Yaskawa INFORM job: blower_cylinder_program.JBI

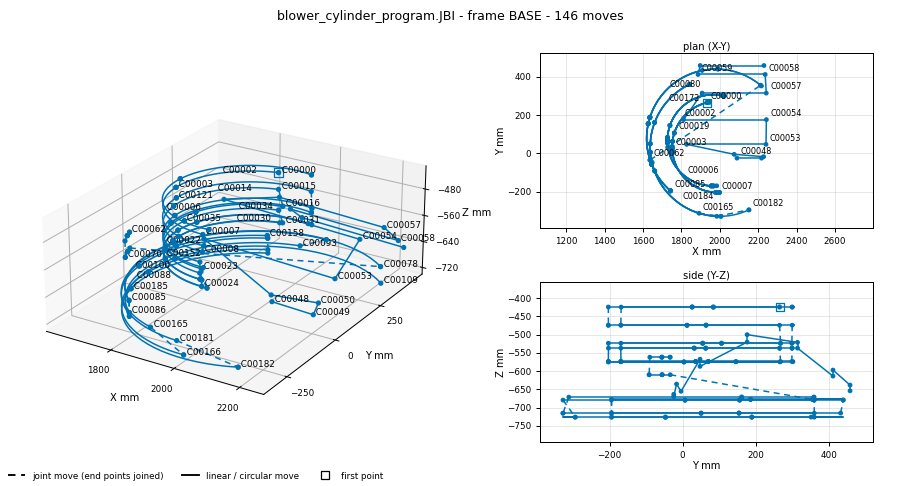
[picture p0: tool path of blower_cylinder_program.JBI in frame BASE, 146 of 201 moves have a stored position in this frame; points joined in program order, loops and branches not executed]
/JOB
//NAME blower_cylinder_program
//POS
///NPOS 190,0,190,0,0,0
///TOOL 0
///POSTYPE BASE
///RECTAN
///RCONF 0,0,0,0,0,0,0,0,0,0,0,0,0,0,0,0,0,0,0,0,0,0,0,0
C00000=1933.494064,265.432065,-424.583000,103.550681,-90.000000,5.000000
C00001=1933.494064,265.432065,-424.583000,103.550681,-90.000000,5.000000
C00002=1798.542139,176.350935,-424.583000,143.306547,-89.999999,5.000000
C00003=1751.564327,26.089320,-424.583000,-175.000000,-90.000000,5.000000
C00004=1751.564327,26.089320,-424.583000,-175.000000,-90.000000,5.000000
C00005=1751.564327,26.089320,-424.583000,-175.000000,-90.000000,5.000000
C00006=1811.478144,-123.700155,-424.583000,-138.369256,-90.000000,5.000000
C00007=1986.712740,-203.504840,-424.583000,-90.601327,-89.999999,5.000000
C00008=1985.205000,-203.484234,-474.602000,-90.964662,-90.000000,5.000000
C00009=1985.205000,-203.484234,-474.602000,-90.964662,-90.000000,5.000000
C00010=1831.755761,-143.919254,-474.602000,-131.465158,-89.999999,5.000000
C00011=1752.467395,12.011979,-474.602000,-174.629726,-90.000000,5.000000
C00012=1752.467395,12.011979,-474.602000,-174.629726,-90.000000,5.000000
C00013=1752.467395,12.011979,-474.602000,-174.629726,-90.000000,5.000000
C00014=1789.907703,163.961680,-474.602000,146.945900,-90.000000,5.000000
C00015=1933.747591,265.493022,-474.602000,103.487851,-90.000000,5.000000
C00016=1946.318295,268.151177,-523.863500,100.391501,-90.000000,5.000000
C00017=1946.318295,268.151177,-523.863500,100.391501,-90.000000,5.000000
C00018=1857.013607,231.918088,-523.863500,123.775687,-90.000000,5.000000
C00019=1762.672230,106.536544,-523.863500,162.306197,-90.000000,5.000000
C00020=1762.672230,106.536544,-523.863500,162.306197,-90.000000,5.000000
C00021=1762.672230,106.536544,-523.863500,162.306197,-90.000000,5.000000
C00022=1803.833605,-114.655285,-523.863500,-141.223119,-90.000000,5.000000
C00023=1981.181892,-203.382432,-523.863500,-91.934378,-90.000000,5.000000
C00024=1982.070197,-203.410772,-573.993000,-91.720226,-89.999999,5.000000
C00025=1982.070197,-203.410772,-573.993000,-91.720226,-89.999999,5.000000
C00026=1827.997866,-140.526698,-573.993000,-132.685079,-90.000000,5.000000
C00027=1751.426860,35.497028,-573.993000,175.000000,-90.000000,5.000000
C00028=1751.426860,35.497028,-573.993000,175.000000,-90.000000,5.000000
C00029=1751.426860,35.497028,-573.993000,175.000000,-90.000000,5.000000
C00030=1823.986848,205.273668,-573.993000,134.014193,-90.000000,5.000000
C00031=1946.357863,268.158430,-573.993000,100.381809,-89.999999,5.000000
C00032=1934.436096,265.657079,-537.267460,175.000000,-60.000000,-76.682693
C00033=1934.436096,265.657079,-537.267460,175.000000,-60.000000,-76.682693
C00034=1828.865200,209.855997,-537.267460,-175.000000,-60.000000,-47.598579
C00035=1753.185183,63.156372,-537.267460,175.000000,-60.000000,-6.978408
C00036=1753.185183,63.156372,-537.267460,175.000000,-60.000000,-6.978408
C00037=1753.185183,63.156372,-537.267460,175.000000,-60.000000,-6.978408
C00038=1809.805430,-121.797856,-537.267460,-175.000000,-60.000000,41.020368
C00039=1976.108054,-203.156798,-537.267460,-175.000000,-60.000000,86.841815
C00040=1998.571162,-203.333530,-575.058960,175.000000,-60.000000,92.256633
C00041=1998.571162,-203.333530,-575.058960,175.000000,-60.000000,92.256633
C00042=1843.618470,-153.736326,-575.058960,175.000000,-60.000000,52.245744
C00043=1753.406955,3.619432,-575.058960,175.000000,-60.000000,7.405254
C00044=1753.406955,3.619432,-575.058960,175.000000,-60.000000,7.405254
C00045=1753.406955,3.619432,-575.058960,175.000000,-60.000000,7.405254
C00046=1795.171150,171.711596,-575.058960,175.000000,-60.000000,-35.311600
C00047=1937.779187,266.423001,-575.058960,-175.000000,-60.000000,-77.509111
C00048=2089.306045,-24.353058,-663.745553,175.000000,-60.000000,90.065286
C00049=2217.470262,-24.353051,-669.800856,175.000000,-60.000000,90.065286
C00050=2228.297277,-16.748565,-635.673601,-175.000000,-60.000000,91.170202
C00051=2074.711330,-4.438705,-655.515790,175.000000,-66.623448,91.170202
C00052=1827.048359,47.582539,-567.652515,175.000000,-44.740427,92.732701
C00053=2240.740165,47.582562,-587.197981,175.000000,-44.740427,92.732701
C00054=2242.656280,176.551574,-520.760389,-170.133186,5.000000,5.000000
C00055=1810.757184,176.551550,-500.354693,-170.133186,5.000000,5.000000
C00056=1907.631611,314.643219,-521.482904,156.457092,5.000000,-5.000000
C00057=2242.006831,314.643237,-537.280944,156.457092,5.000000,-5.000000
C00058=2236.445037,411.851577,-613.890742,175.000000,-53.159924,-92.028486
C00059=1886.225138,411.851557,-597.344097,175.000000,-53.159924,-92.028486
C00060=1897.676258,458.517871,-638.458617,175.000000,-60.000000,-90.549119
C00061=2229.933616,458.517890,-654.156596,175.000000,-60.000000,-90.549119
C00062=1636.254154,-34.391820,-562.117000,-161.880193,-90.000000,5.000000
C00063=1636.254154,-34.391820,-562.117000,-161.880193,-90.000000,5.000000
C00064=1640.360805,-46.242627,-562.117000,-159.894424,-89.999999,5.000000
C00065=1644.466194,-56.930864,-562.117000,-158.081660,-90.000000,5.000000
C00066=1644.466194,-56.930864,-562.117000,-158.081660,-90.000000,5.000000
C00067=1644.466194,-56.930864,-562.117000,-158.081660,-90.000000,5.000000
C00068=1652.539385,-75.480262,-562.117000,-154.878428,-90.000000,5.000000
C00069=1659.732185,-89.968706,-562.117000,-152.317297,-89.999999,5.000000
C00070=1660.669780,-91.743887,-610.141500,-151.999459,-90.000000,5.000000
C00071=1660.669780,-91.743887,-610.141500,-151.999459,-90.000000,5.000000
C00072=1649.493547,-68.809454,-610.141500,-156.039446,-89.999999,5.000000
C00073=1644.226079,-56.332574,-610.141500,-158.183725,-90.000000,5.000000
C00074=1644.226079,-56.332574,-610.141500,-158.183725,-90.000000,5.000000
C00075=1644.226079,-56.332574,-610.141500,-158.183725,-90.000000,5.000000
C00076=1639.543696,-43.987319,-610.141500,-160.274196,-89.999999,5.000000
C00077=1636.130097,-34.012000,-610.141500,-161.943452,-90.000000,5.000000
C00078=2212.617724,355.571818,-677.762000,50.044218,-90.000000,5.000000
C00079=2212.617724,355.571818,-677.762000,50.044218,-90.000000,5.000000
C00080=1718.993255,328.638505,-677.762000,136.201974,-90.000000,5.000000
C00081=1634.749633,186.007445,-677.762000,162.662423,-90.000000,5.000000
C00082=1634.749633,186.007445,-677.762000,162.662423,-90.000000,5.000000
C00083=1634.749633,186.007445,-677.762000,162.662423,-90.000000,5.000000
C00084=1619.374320,50.385855,-677.762000,-175.000000,-90.000000,5.000000
C00085=1742.557948,-194.776065,-677.762000,-131.046419,-90.000000,5.000000
C00086=1742.571134,-194.787546,-715.259500,-131.043651,-89.999999,5.000000
C00087=1742.571134,-194.787546,-715.259500,-131.043651,-89.999999,5.000000
C00088=1627.706250,-3.783572,-715.259500,-166.913109,-89.999999,5.000000
C00089=1626.423323,154.376268,-715.259500,167.842607,-90.000000,5.000000
C00090=1626.423323,154.376268,-715.259500,167.842607,-90.000000,5.000000
C00091=1626.423323,154.376268,-715.259500,167.842607,-90.000000,5.000000
C00092=1698.604915,305.475486,-715.259500,141.088858,-90.000000,5.000000
C00093=1907.554137,432.693235,-715.259500,101.581038,-90.000000,5.000000
C00094=1990.113591,439.925270,-679.410460,-175.000000,-60.000000,-91.568615
C00095=1990.113591,439.925270,-679.410460,-175.000000,-60.000000,-91.568615
C00096=1716.864165,326.399098,-679.410460,175.000000,-60.000000,-43.308821
C00097=1626.783413,156.028994,-679.410460,175.000000,-60.000000,-12.425190
C00098=1626.783413,156.028994,-679.410460,175.000000,-60.000000,-12.425190
C00099=1626.783413,156.028994,-679.410460,175.000000,-60.000000,-12.425190
C00100=1629.721714,-12.015259,-679.410460,175.000000,-60.000000,14.428652
C00101=1742.946883,-195.114229,-679.410460,-175.000000,-60.000000,49.035177
C00102=1742.486630,-194.713952,-726.158960,175.000000,-60.000000,48.938608
C00103=1742.486630,-194.713952,-726.158960,175.000000,-60.000000,48.938608
C00104=1625.571685,6.011963,-726.158960,-175.000000,-60.000000,11.499624
C00105=1635.832274,189.416091,-726.158960,175.000000,-60.000000,-17.903800
C00106=1635.832274,189.416091,-726.158960,175.000000,-60.000000,-17.903800
C00107=1635.832274,189.416091,-726.158960,175.000000,-60.000000,-17.903800
C00108=1743.075199,351.547358,-726.158960,-175.000000,-60.000000,-49.062075
C00109=2217.001537,351.839376,-726.158960,175.000000,-60.000000,-130.867317
C00110=2018.613598,300.043424,-424.810500,76.870993,-90.000000,5.000000
C00111=2018.613598,300.043424,-424.810500,76.870993,-90.000000,5.000000
C00112=1820.893884,257.919353,-424.810500,127.183038,-89.999999,5.000000
C00113=1727.333238,84.125835,-424.810500,175.000000,-90.000000,5.000000
C00114=1727.333238,84.125835,-424.810500,175.000000,-90.000000,5.000000
C00115=1727.333238,84.125835,-424.810500,175.000000,-90.000000,5.000000
C00116=1798.162352,-101.347137,-424.810500,-134.423830,-90.000000,5.000000
C00117=1983.786314,-168.535208,-424.810500,-85.372422,-90.000000,5.000000
C00118=1967.525308,-169.292379,-474.431000,-89.295632,-90.000000,5.000000
C00119=1967.525308,-169.292379,-474.431000,-89.295632,-90.000000,5.000000
C00120=1803.643952,-106.551373,-474.431000,-132.602465,-90.000000,5.000000
C00121=1726.858274,64.074444,-474.431000,-175.000000,-89.999999,5.000000
C00122=1726.858274,64.074444,-474.431000,-175.000000,-89.999999,5.000000
C00123=1726.858274,64.074444,-474.431000,-175.000000,-89.999999,5.000000
C00124=1799.110942,239.220178,-474.431000,134.104657,-90.000000,5.000000
C00125=2018.648093,300.035376,-474.431000,76.862458,-89.999999,5.000000
C00126=2022.017279,299.223079,-523.805000,76.027362,-90.000000,5.000000
C00127=2022.017279,299.223079,-523.805000,76.027362,-90.000000,5.000000
C00128=1811.476704,250.392117,-523.805000,130.088277,-90.000000,5.000000
C00129=1727.204719,54.910761,-523.805000,-175.000000,-90.000000,5.000000
C00130=1727.204719,54.910761,-523.805000,-175.000000,-90.000000,5.000000
C00131=1727.204719,54.910761,-523.805000,-175.000000,-90.000000,5.000000
C00132=1877.695238,-152.859662,-523.805000,-111.437491,-89.999999,5.000000
C00133=1954.764997,-169.106778,-523.805000,-92.371008,-89.999999,5.000000
C00134=1954.809816,-169.108629,-573.819000,-92.360199,-90.000000,5.000000
C00135=1954.809816,-169.108629,-573.819000,-92.360199,-90.000000,5.000000
C00136=1838.292406,-132.988797,-573.819000,-122.086166,-89.999999,5.000000
C00137=1726.823702,70.182652,-573.819000,175.000000,-89.999999,5.000000
C00138=1726.823702,70.182652,-573.819000,175.000000,-89.999999,5.000000
C00139=1726.823702,70.182652,-573.819000,175.000000,-89.999999,5.000000
C00140=1810.644481,249.688346,-573.819000,130.350897,-90.000000,5.000000
C00141=2022.320648,299.147383,-573.819000,75.952022,-90.000000,5.000000
C00142=2020.266527,299.651663,-537.232460,175.000000,-60.000000,-103.538326
C00143=2020.266527,299.651663,-537.232460,175.000000,-60.000000,-103.538326
C00144=1793.642119,233.744271,-537.232460,-175.000000,-60.000000,-44.030475
C00145=1729.658981,31.824341,-537.232460,175.000000,-60.000000,8.866385
C00146=1729.658981,31.824341,-537.232460,175.000000,-60.000000,8.866385
C00147=1729.658981,31.824341,-537.232460,175.000000,-60.000000,8.866385
C00148=1882.234966,-154.588878,-537.232460,-175.000000,-60.000000,69.733076
C00149=1965.409561,-169.308976,-537.232460,175.000000,-60.000000,90.194548
C00150=1960.148078,-169.268627,-574.430960,175.000000,-60.000000,88.926695
C00151=1960.148078,-169.268627,-574.430960,175.000000,-60.000000,88.926695
C00152=1789.870915,-92.803477,-574.430960,-175.000000,-60.000000,42.707149
C00153=1739.810945,146.001172,-574.430960,-175.000000,-60.000000,-19.028500
C00154=1739.810945,146.001172,-574.430960,-175.000000,-60.000000,-19.028500
C00155=1739.810945,146.001172,-574.430960,-175.000000,-60.000000,-19.028500
C00156=1871.976480,287.476533,-574.430960,-175.000000,-60.000000,-67.074363
C00157=2009.127801,302.052899,-574.430960,-175.000000,-60.000000,-100.792456
C00158=1840.845613,359.624038,-671.548000,115.867977,-89.999999,5.000000
C00159=1840.845613,359.624038,-671.548000,115.867977,-89.999999,5.000000
C00160=1750.456884,297.284107,-671.548000,133.319072,-89.999999,5.000000
C00161=1660.063951,161.534400,-671.548000,159.363272,-90.000000,5.000000
C00162=1660.063951,161.534400,-671.548000,159.363272,-90.000000,5.000000
C00163=1660.063951,161.534400,-671.548000,159.363272,-90.000000,5.000000
C00164=1663.681234,-102.783213,-671.548000,-157.795142,-90.000000,5.000000
C00165=1892.003030,-311.815262,-671.548000,-107.154004,-90.000000,5.000000
C00166=2005.541885,-327.850338,-715.502500,-88.923415,-89.999999,5.000000
C00167=2005.541885,-327.850338,-715.502500,-88.923415,-89.999999,5.000000
C00168=1716.504333,-192.538822,-715.502500,-141.249412,-89.999999,5.000000
C00169=1637.218632,50.487820,-715.502500,175.000000,-90.000000,5.000000
C00170=1637.218632,50.487820,-715.502500,175.000000,-90.000000,5.000000
C00171=1637.218632,50.487820,-715.502500,175.000000,-90.000000,5.000000
C00172=1710.989194,253.462007,-715.502500,142.666352,-90.000000,5.000000
C00173=1842.663843,360.499415,-715.502500,115.548491,-89.999999,5.000000
C00174=1842.194123,360.274466,-679.645460,175.000000,-60.000000,-64.369055
C00175=1842.194123,360.274466,-679.645460,175.000000,-60.000000,-64.369055
C00176=1707.789251,249.201923,-679.645460,175.000000,-60.000000,-36.490110
C00177=1637.882326,6.567565,-679.645460,175.000000,-60.000000,5.000000
C00178=1637.882326,6.567565,-679.645460,175.000000,-60.000000,5.000000
C00179=1637.882326,6.567565,-679.645460,175.000000,-60.000000,5.000000
C00180=1702.234553,-173.510785,-679.645460,175.000000,-60.000000,34.984395
C00181=1984.418511,-327.630652,-679.645460,-175.000000,-60.000000,87.731690
C00182=2151.462989,-294.111726,-726.328460,175.000000,-60.000000,114.960743
C00183=2151.462989,-294.111726,-726.328460,175.000000,-60.000000,114.960743
C00184=1784.065592,-257.365492,-726.328460,175.000000,-60.000000,53.616065
C00185=1646.036132,-47.069987,-726.328460,175.000000,-60.000000,12.942484
C00186=1646.036132,-47.069987,-726.328460,175.000000,-60.000000,12.942484
C00187=1646.036132,-47.069987,-726.328460,175.000000,-60.000000,12.942484
C00188=1687.963593,219.426510,-726.328460,175.000000,-60.000000,-30.824410
C00189=1842.566553,360.452891,-726.328460,-175.000000,-60.000000,-64.434435
///POSTYPE PULSE
///PULSE
EX00000=40960.0
EX00001=113664.0
EX00002=115712.0
EX00003=212992.0
EX00004=368640.0
///POSTYPE PULSE
///PULSE
EC00000=40960.0
EC00001=40960.0
EC00002=40960.0
EC00003=40960.0
EC00004=40960.0
EC00005=40960.0
EC00006=40960.0
EC00007=40960.0
EC00008=40960.0
EC00009=40960.0
EC00010=40960.0
EC00011=40960.0
EC00012=40960.0
EC00013=40960.0
EC00014=40960.0
EC00015=40960.0
EC00016=40960.0
EC00017=40960.0
EC00018=40960.0
EC00019=40960.0
EC00020=40960.0
EC00021=40960.0
EC00022=40960.0
EC00023=40960.0
EC00024=40960.0
EC00025=40960.0
EC00026=40960.0
EC00027=40960.0
EC00028=40960.0
EC00029=40960.0
EC00030=40960.0
EC00031=40960.0
EC00032=40960.0
EC00033=40960.0
EC00034=40960.0
EC00035=40960.0
EC00036=40960.0
EC00037=40960.0
EC00038=40960.0
EC00039=40960.0
EC00040=40960.0
EC00041=40960.0
EC00042=40960.0
EC00043=40960.0
EC00044=40960.0
EC00045=40960.0
EC00046=40960.0
EC00047=40960.0
EC00048=113664.0
EC00049=113664.0
EC00050=113664.0
EC00051=113664.0
EC00052=113664.0
EC00053=113664.0
EC00054=113664.0
EC00055=113664.0
EC00056=113664.0
EC00057=113664.0
EC00058=113664.0
EC00059=113664.0
EC00060=113664.0
EC00061=113664.0
EC00062=115712.0
EC00063=115712.0
EC00064=115712.0
EC00065=115712.0
EC00066=115712.0
EC00067=115712.0
EC00068=115712.0
EC00069=115712.0
EC00070=115712.0
EC00071=115712.0
EC00072=115712.0
EC00073=115712.0
EC00074=115712.0
EC00075=115712.0
EC00076=115712.0
EC00077=115712.0
EC00078=115712.0
EC00079=115712.0
EC00080=115712.0
EC00081=115712.0
EC00082=115712.0
EC00083=115712.0
EC00084=115712.0
EC00085=115712.0
EC00086=115712.0
EC00087=115712.0
EC00088=115712.0
EC00089=115712.0
EC00090=115712.0
EC00091=115712.0
EC00092=115712.0
EC00093=115712.0
EC00094=115712.0
EC00095=115712.0
EC00096=115712.0
EC00097=115712.0
EC00098=115712.0
EC00099=115712.0
EC00100=115712.0
EC00101=115712.0
EC00102=115712.0
EC00103=115712.0
EC00104=115712.0
EC00105=115712.0
EC00106=115712.0
EC00107=115712.0
EC00108=115712.0
EC00109=115712.0
EC00110=212992.0
EC00111=212992.0
EC00112=212992.0
EC00113=212992.0
EC00114=212992.0
EC00115=212992.0
EC00116=212992.0
EC00117=212992.0
EC00118=212992.0
EC00119=212992.0
EC00120=212992.0
EC00121=212992.0
EC00122=212992.0
EC00123=212992.0
EC00124=212992.0
EC00125=212992.0
EC00126=212992.0
EC00127=212992.0
EC00128=212992.0
EC00129=212992.0
EC00130=212992.0
EC00131=212992.0
EC00132=212992.0
EC00133=212992.0
EC00134=212992.0
EC00135=212992.0
EC00136=212992.0
EC00137=212992.0
EC00138=212992.0
EC00139=212992.0
EC00140=212992.0
EC00141=212992.0
EC00142=212992.0
EC00143=212992.0
EC00144=212992.0
EC00145=212992.0
EC00146=212992.0
EC00147=212992.0
EC00148=212992.0
EC00149=212992.0
EC00150=212992.0
EC00151=212992.0
EC00152=212992.0
EC00153=212992.0
EC00154=212992.0
EC00155=212992.0
EC00156=212992.0
EC00157=212992.0
EC00158=368640.0
EC00159=368640.0
EC00160=368640.0
EC00161=368640.0
EC00162=368640.0
EC00163=368640.0
EC00164=368640.0
EC00165=368640.0
EC00166=368640.0
EC00167=368640.0
EC00168=368640.0
EC00169=368640.0
EC00170=368640.0
EC00171=368640.0
EC00172=368640.0
EC00173=368640.0
EC00174=368640.0
EC00175=368640.0
EC00176=368640.0
EC00177=368640.0
EC00178=368640.0
EC00179=368640.0
EC00180=368640.0
EC00181=368640.0
EC00182=368640.0
EC00183=368640.0
EC00184=368640.0
EC00185=368640.0
EC00186=368640.0
EC00187=368640.0
EC00188=368640.0
EC00189=368640.0
//INST
///DATE 2023/08/15 16:25
///ATTR SC,RW,RJ
////FRAME BASE
///GROUP1 RB1,ST1
NOP
MOVJ P009 EX000 VJ=15.00
MOVJ C00000 EC00000 VJ=15.0
CALL JOB:SPYON
MOVC C00001 EC00001 V=150.0
MOVC C00002 EC00002 V=150.0
MOVC C00003 EC00003 V=150.0
MOVJ C00004 EC00004 VJ=15.0
MOVC C00005 EC00005 V=150.0
MOVC C00006 EC00006 V=150.0
MOVC C00007 EC00007 V=150.0
MOVJ C00008 EC00008 VJ=15.0
MOVC C00009 EC00009 V=150.0
MOVC C00010 EC00010 V=150.0
MOVC C00011 EC00011 V=150.0
MOVJ C00012 EC00012 VJ=15.0
MOVC C00013 EC00013 V=150.0
MOVC C00014 EC00014 V=150.0
MOVC C00015 EC00015 V=150.0
MOVJ C00016 EC00016 VJ=15.0
MOVC C00017 EC00017 V=150.0
MOVC C00018 EC00018 V=150.0
MOVC C00019 EC00019 V=150.0
MOVJ C00020 EC00020 VJ=15.0
MOVC C00021 EC00021 V=150.0
MOVC C00022 EC00022 V=150.0
MOVC C00023 EC00023 V=150.0
MOVJ C00024 EC00024 VJ=15.0
MOVC C00025 EC00025 V=150.0
MOVC C00026 EC00026 V=150.0
MOVC C00027 EC00027 V=150.0
MOVJ C00028 EC00028 VJ=15.0
MOVC C00029 EC00029 V=150.0
MOVC C00030 EC00030 V=150.0
MOVC C00031 EC00031 V=150.0
MOVJ C00032 EC00032 VJ=15.0
MOVC C00033 EC00033 V=150.0
MOVC C00034 EC00034 V=150.0
MOVC C00035 EC00035 V=150.0
MOVJ C00036 EC00036 VJ=15.0
MOVC C00037 EC00037 V=150.0
MOVC C00038 EC00038 V=150.0
MOVC C00039 EC00039 V=150.0
MOVJ C00040 EC00040 VJ=15.0
MOVC C00041 EC00041 V=150.0
MOVC C00042 EC00042 V=150.0
MOVC C00043 EC00043 V=150.0
MOVJ C00044 EC00044 VJ=15.0
MOVC C00045 EC00045 V=150.0
MOVC C00046 EC00046 V=150.0
MOVC C00047 EC00047 V=150.0
CALL JOB:SPYOF
MOVJ P009 VJ=15.00
MOVL P009 EX00000 V=150.0
MOVJ C00048 EC00048 VJ=15.0
CALL JOB:SPYON
MOVL C00049 EC00049 V=150.0
MOVL C00050 EC00050 V=150.0
MOVL C00051 EC00051 V=150.0
MOVL C00052 EC00052 V=150.0
MOVL C00053 EC00053 V=150.0
MOVL C00054 EC00054 V=150.0
MOVL C00055 EC00055 V=150.0
MOVL C00056 EC00056 V=150.0
MOVL C00057 EC00057 V=150.0
MOVL C00058 EC00058 V=150.0
MOVL C00059 EC00059 V=150.0
MOVL C00060 EC00060 V=150.0
MOVL C00061 EC00061 V=150.0
CALL JOB:SPYOF
MOVJ P009 VJ=15.00
MOVL P009 EX00001 V=150.0
MOVJ C00062 EC00062 VJ=15.0
CALL JOB:SPYON
MOVC C00063 EC00063 V=150.0
MOVC C00064 EC00064 V=150.0
MOVC C00065 EC00065 V=150.0
MOVJ C00066 EC00066 VJ=15.0
MOVC C00067 EC00067 V=150.0
MOVC C00068 EC00068 V=150.0
MOVC C00069 EC00069 V=150.0
MOVJ C00070 EC00070 VJ=15.0
MOVC C00071 EC00071 V=150.0
MOVC C00072 EC00072 V=150.0
MOVC C00073 EC00073 V=150.0
MOVJ C00074 EC00074 VJ=15.0
MOVC C00075 EC00075 V=150.0
MOVC C00076 EC00076 V=150.0
MOVC C00077 EC00077 V=150.0
MOVJ C00078 EC00078 VJ=15.0
MOVC C00079 EC00079 V=150.0
MOVC C00080 EC00080 V=150.0
MOVC C00081 EC00081 V=150.0
MOVJ C00082 EC00082 VJ=15.0
MOVC C00083 EC00083 V=150.0
MOVC C00084 EC00084 V=150.0
MOVC C00085 EC00085 V=150.0
MOVJ C00086 EC00086 VJ=15.0
MOVC C00087 EC00087 V=150.0
MOVC C00088 EC00088 V=150.0
MOVC C00089 EC00089 V=150.0
MOVJ C00090 EC00090 VJ=15.0
MOVC C00091 EC00091 V=150.0
MOVC C00092 EC00092 V=150.0
MOVC C00093 EC00093 V=150.0
MOVJ C00094 EC00094 VJ=15.0
MOVC C00095 EC00095 V=150.0
MOVC C00096 EC00096 V=150.0
MOVC C00097 EC00097 V=150.0
MOVJ C00098 EC00098 VJ=15.0
MOVC C00099 EC00099 V=150.0
MOVC C00100 EC00100 V=150.0
MOVC C00101 EC00101 V=150.0
MOVJ C00102 EC00102 VJ=15.0
MOVC C00103 EC00103 V=150.0
MOVC C00104 EC00104 V=150.0
MOVC C00105 EC00105 V=150.0
MOVJ C00106 EC00106 VJ=15.0
MOVC C00107 EC00107 V=150.0
MOVC C00108 EC00108 V=150.0
MOVC C00109 EC00109 V=150.0
CALL JOB:SPYOF
MOVJ P009 VJ=15.00
MOVL P009 EX00002 V=150.0
MOVJ C00110 EC00110 VJ=15.0
CALL JOB:SPYON
MOVC C00111 EC00111 V=150.0
MOVC C00112 EC00112 V=150.0
MOVC C00113 EC00113 V=150.0
MOVJ C00114 EC00114 VJ=15.0
MOVC C00115 EC00115 V=150.0
MOVC C00116 EC00116 V=150.0
MOVC C00117 EC00117 V=150.0
MOVJ C00118 EC00118 VJ=15.0
MOVC C00119 EC00119 V=150.0
MOVC C00120 EC00120 V=150.0
MOVC C00121 EC00121 V=150.0
MOVJ C00122 EC00122 VJ=15.0
MOVC C00123 EC00123 V=150.0
MOVC C00124 EC00124 V=150.0
MOVC C00125 EC00125 V=150.0
MOVJ C00126 EC00126 VJ=15.0
MOVC C00127 EC00127 V=150.0
MOVC C00128 EC00128 V=150.0
MOVC C00129 EC00129 V=150.0
MOVJ C00130 EC00130 VJ=15.0
MOVC C00131 EC00131 V=150.0
MOVC C00132 EC00132 V=150.0
MOVC C00133 EC00133 V=150.0
MOVJ C00134 EC00134 VJ=15.0
MOVC C00135 EC00135 V=150.0
MOVC C00136 EC00136 V=150.0
MOVC C00137 EC00137 V=150.0
MOVJ C00138 EC00138 VJ=15.0
MOVC C00139 EC00139 V=150.0
MOVC C00140 EC00140 V=150.0
MOVC C00141 EC00141 V=150.0
MOVJ C00142 EC00142 VJ=15.0
MOVC C00143 EC00143 V=150.0
MOVC C00144 EC00144 V=150.0
MOVC C00145 EC00145 V=150.0
MOVJ C00146 EC00146 VJ=15.0
MOVC C00147 EC00147 V=150.0
MOVC C00148 EC00148 V=150.0
MOVC C00149 EC00149 V=150.0
MOVJ C00150 EC00150 VJ=15.0
MOVC C00151 EC00151 V=150.0
MOVC C00152 EC00152 V=150.0
MOVC C00153 EC00153 V=150.0
MOVJ C00154 EC00154 VJ=15.0
MOVC C00155 EC00155 V=150.0
MOVC C00156 EC00156 V=150.0
MOVC C00157 EC00157 V=150.0
CALL JOB:SPYOF
MOVJ P009 VJ=15.00
MOVL P009 EX00003 V=150.0
MOVJ C00158 EC00158 VJ=15.0
CALL JOB:SPYON
MOVC C00159 EC00159 V=150.0
MOVC C00160 EC00160 V=150.0
MOVC C00161 EC00161 V=150.0
MOVJ C00162 EC00162 VJ=15.0
MOVC C00163 EC00163 V=150.0
MOVC C00164 EC00164 V=150.0
MOVC C00165 EC00165 V=150.0
MOVJ C00166 EC00166 VJ=15.0
MOVC C00167 EC00167 V=150.0
MOVC C00168 EC00168 V=150.0
MOVC C00169 EC00169 V=150.0
MOVJ C00170 EC00170 VJ=15.0
MOVC C00171 EC00171 V=150.0
MOVC C00172 EC00172 V=150.0
MOVC C00173 EC00173 V=150.0
MOVJ C00174 EC00174 VJ=15.0
MOVC C00175 EC00175 V=150.0
MOVC C00176 EC00176 V=150.0
MOVC C00177 EC00177 V=150.0
MOVJ C00178 EC00178 VJ=15.0
MOVC C00179 EC00179 V=150.0
MOVC C00180 EC00180 V=150.0
MOVC C00181 EC00181 V=150.0
MOVJ C00182 EC00182 VJ=15.0
MOVC C00183 EC00183 V=150.0
MOVC C00184 EC00184 V=150.0
MOVC C00185 EC00185 V=150.0
MOVJ C00186 EC00186 VJ=15.0
MOVC C00187 EC00187 V=150.0
MOVC C00188 EC00188 V=150.0
MOVC C00189 EC00189 V=150.0
CALL JOB:SPYOF
MOVJ P009 VJ=15.00
MOVL P009 EX00004 V=150.0
END
